/// calibration that is determined by calibration sequences of the unit (static offsets, shifts)
TYPE HandlingDataCalibration :
STRUCT
END_STRUCT
END_TYPE

(* stored: Version 1.1.0.1
   DUT HandlingDataCalibration: Id {5cc061e7-647e-427f-80b5-a2e13760b1ad} *)
